{region '#Template'}
	{attribute 'Version' := '1.2.2.0'}
	{attribute 'Tags' := '"LCID": "1031", "Text": "Universal, Control, Monitoring"'}
	{attribute 'Tags' := '"LCID": "1033", "Text": "Universal, Control, Monitoring"'}
	{attribute 'Using' := '"Type": "Template", "URI": "EC_AMEV"'}
	{attribute 'Using' := '"Type": "Template", "URI": "BA2_Param"'}
	{attribute 'Description' := '"LCID": "1031", "Text": "Überwachung von Signalen"'}
	{attribute 'Description' := '"LCID": "1033", "Text": "Monitoring signals"'}
{endregion}
FUNCTION_BLOCK FB_BA_FdbBinary EXTENDS FB_BA_View
VAR_INPUT
	bEn						: BOOL;	
	bCommand				: BOOL;	
	bFeedback				: BOOL;		
END_VAR
VAR_OUTPUT
	bDst					: BOOL;
END_VAR
VAR_INPUT CONSTANT
	DelayFeedback			: FB_BA_AV_Op;
	Dst						: FB_BA_BV;			
END_VAR
VAR_INPUT CONSTANT PERSISTENT
	{attribute 'parameterUnit':= 's'}
	nInterruptionDelay : UDINT := 1;
END_VAR
VAR
	FdbCtrl					: FB_BA_FdbCtrlBinary;		
END_VAR

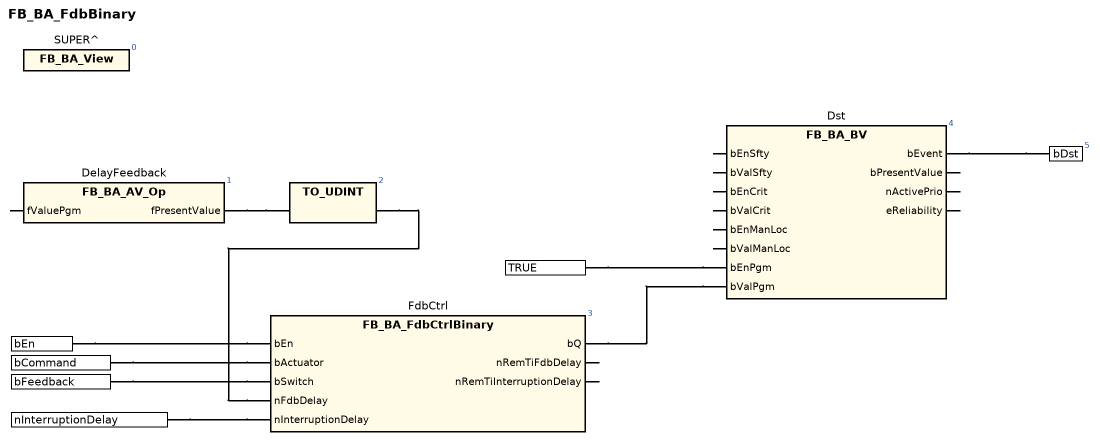
SUPER^(); // FB_BA_View
DelayFeedback(); // FB_BA_AV_Op
FdbCtrl(
    bEn := bEn,
    bActuator := bCommand,
    bSwitch := bFeedback,
    nFdbDelay := TO_UDINT(DelayFeedback.fPresentValue),
    nInterruptionDelay := nInterruptionDelay); // FB_BA_FdbCtrlBinary
Dst(bEnPgm := TRUE, bValPgm := FdbCtrl.bQ); // FB_BA_BV
bDst := Dst.bEvent;

METHOD FB_init : BOOL
VAR_INPUT
	bInitRetains : BOOL; // if TRUE, the retain variables are initialized (warm start / cold start)
	bInCopyCode : BOOL;  // if TRUE, the instance afterwards gets moved into the copy code (online change)
END_VAR
DelayFeedback.iParent				:= THIS^;
DelayFeedback.iLabel				:= LblUniControl.Monitoring_DelayFeedback;	 								 
DelayFeedback.sObjectName			:= '{Idx=01}';								 	 
DelayFeedback.eUnit 				:= E_BA_Unit.eTime_Seconds;								 
DelayFeedback.fValueRm 				:= 120;
DelayFeedback.fCOVIncrement			:= BA2_Param.fDefCOVIncrement;		

Dst.iParent							:= THIS^;
Dst.iLabel							:= LblUniControl.Monitoring_Dst;			
Dst.sObjectName						:= '{Idx=01}';	
Dst.bEnOutOfService					:= FALSE;
Dst.sActiveText 					:= txtEvent_Triggered;
Dst.sInactiveText 					:= txtEvent_Normal;
Dst.nStateChangeCount				:= 0;
Dst.nActiveTimeElapsed				:= 0;
Dst.nMinimumOnTime					:= 0;
Dst.nMinimumOffTime					:= 0;
Dst.bEnManualRm						:= FALSE;	//	Priority  8	
Dst.bValManualRm					:= FALSE;	//	Priority  8
Dst.bDefaultValue					:= FALSE;
Dst.nEventClassID					:= EC_ID.NC30;
Dst.stTimeDelay.nToNormal			:= 0;
Dst.stTimeDelay.nToAbnormal			:= 0;
Dst.bAlarmValue						:= TRUE;
Dst.bAcknowledgeRm					:= FALSE;		
Dst.aEventTransitionText[1]			:= txtEvent_Triggered;
Dst.aEventTransitionText[2]			:= txtEvent_Error;
Dst.aEventTransitionText[3]			:= txtEvent_Normal;
Dst.bEventDetectionEnable			:= TRUE;
Dst.aEventEnable[1]					:= TRUE;			//	to_offnormal
Dst.aEventEnable[2]					:= TRUE;			//	to_fault
Dst.aEventEnable[3]					:= TRUE;			//	to_normal
Dst.eEnPlantLock					:= E_BA_LockPriority.eNoLock;
END_METHOD

END_FUNCTION_BLOCK

(* stored: Version 1.1.0.1, ProductVersion 3.1.4024.9
   POU FB_BA_FdbBinary: Id {b776b9c7-cfde-4809-be07-b3ebe0c5346f}, SpecialFunc None
   Method FB_init: Id {04d8e280-50f3-4c89-b4bb-5d13216e2285} *)
